// TIA Portal project "PLC_Working" (V16)

(* hardware
DEVICE "S71500/ET200MP station_1"  S7-1500 station
   slot 0: "Rail_0"  Rack  6ES7 590-1***0-0AA0
   slot 1: "PLC_1"  CPU 1515-2 PN  6ES7 515-2AM02-0AB0  V2.8
      slot 3: "CPU display_1"  6ES7591-1BA00-0AA0
      slot 32768: "PROFINET interface_1"  X1
         slot 32769: "Port_1"  X1 P1
         slot 32770: "Port_2"  X1 P2
      slot 33024: "PROFINET interface_2"  X2
      slot 34817: "Virtual CP interface port_1"  Virtual CP interface port  Virtual CP interface port
*)

// ===== PLC "PLC_1"  CPU 1515-2 PN =====

VAR_GLOBAL   // PLC tag table "Default tag table"
   "System_Byte" AT %MB1 : Byte;
   "FirstScan" AT %M1.0 : Bool;
   "DiagStatusUpdate" AT %M1.1 : Bool;
   "AlwaysTRUE" AT %M1.2 : Bool;
   "AlwaysFALSE" AT %M1.3 : Bool;
   "Clock_Byte" AT %MB0 : Byte;
   "Clock_10Hz" AT %M0.0 : Bool;
   "Clock_5Hz" AT %M0.1 : Bool;
   "Clock_2.5Hz" AT %M0.2 : Bool;
   "Clock_2Hz" AT %M0.3 : Bool;
   "Clock_1.25Hz" AT %M0.4 : Bool;
   "Clock_1Hz" AT %M0.5 : Bool;
   "Clock_0.625Hz" AT %M0.6 : Bool;
   "Clock_0.5Hz" AT %M0.7 : Bool;
   "in1" AT %M2.0 : Bool;
   "out1" AT %M2.1 : Bool;
   "out2" AT %M2.2 : Bool;
   "out3" AT %M2.3 : Bool;
   "out3_count" AT %MW4 : Int;
   "out1_count" AT %MW6 : Int;
   "T1_OUT" AT %M2.4 : Bool;
   "T2_OUT" AT %M2.5 : Bool;
   "T3_OUT" AT %M2.6 : Bool;
   "T4_OUT" AT %M2.7 : Bool;
   "ET1" AT %MD8 : Time;
   "ET2" AT %MD12 : Time;
   "ET3" AT %MD16 : DWord;
   "ET4" AT %MD20 : DInt;
   "TIMER_SWITCH" AT %M3.0 : Bool;
   "T4_RESET" AT %M3.1 : Bool;
   "in1 timer" AT %M3.2 : Bool;
END_VAR

DATA_BLOCK "LADDER2_DB"   // DB1
{ S7_Optimized_Access := 'TRUE' }
VERSION : 0.1
// stored: InstanceOfName LADDER2
"LADDER2"
BEGIN
END_DATA_BLOCK

DATA_BLOCK "TIMER_OPERATION_DB"   // DB8
{ S7_Optimized_Access := 'TRUE' }
VERSION : 0.1
// stored: InstanceOfName TIMER_OPERATION
"TIMER_OPERATION"
BEGIN
END_DATA_BLOCK

// folder: System blocks/Program resources

DATA_BLOCK "PULSE_TIMER"   // DB2
{ S7_Optimized_Access := 'TRUE' }
AUTHOR : Simatic
FAMILY : IEC
NAME : IEC_TMR
VERSION : 1.0
// stored: InstanceOfName IEC_TIMER
"IEC_TIMER"
BEGIN
END_DATA_BLOCK

DATA_BLOCK "IEC_Counter_0_DB"   // DB3
{ S7_Optimized_Access := 'TRUE' }
AUTHOR : Simatic
FAMILY : IEC
NAME : CNTR
VERSION : 1.0
// stored: InstanceOfName IEC_COUNTER
"IEC_COUNTER"
BEGIN
END_DATA_BLOCK

DATA_BLOCK "IEC_Counter_0_DB_1"   // DB4
{ S7_Optimized_Access := 'TRUE' }
AUTHOR : Simatic
FAMILY : IEC
NAME : CNTR
VERSION : 1.0
// stored: InstanceOfName IEC_COUNTER
"IEC_COUNTER"
BEGIN
END_DATA_BLOCK

DATA_BLOCK "TON_TIMER"   // DB5
{ S7_Optimized_Access := 'TRUE' }
AUTHOR : Simatic
FAMILY : IEC
NAME : IEC_TMR
VERSION : 1.0
// stored: InstanceOfName IEC_TIMER
"IEC_TIMER"
BEGIN
END_DATA_BLOCK

DATA_BLOCK "TOF_TIMER"   // DB6
{ S7_Optimized_Access := 'TRUE' }
AUTHOR : Simatic
FAMILY : IEC
NAME : IEC_TMR
VERSION : 1.0
// stored: InstanceOfName IEC_TIMER
"IEC_TIMER"
BEGIN
END_DATA_BLOCK

DATA_BLOCK "TONR_TIMER"   // DB7
{ S7_Optimized_Access := 'TRUE' }
AUTHOR : Simatic
FAMILY : IEC
NAME : IEC_TMR
VERSION : 1.0
// stored: InstanceOfName IEC_TIMER
"IEC_TIMER"
BEGIN
END_DATA_BLOCK

// folder: (top level)

FUNCTION_BLOCK "LADDER2"   // FB1, LAD
{ S7_Optimized_Access := 'TRUE' }
VERSION : 0.1
   VAR
      ons : Bool;
   END_VAR
   VAR_TEMP   // added for the SCL form of the ladder/FBD networks
      _w1 : Bool;
   END_VAR
BEGIN

REGION Network 1: device 1 control
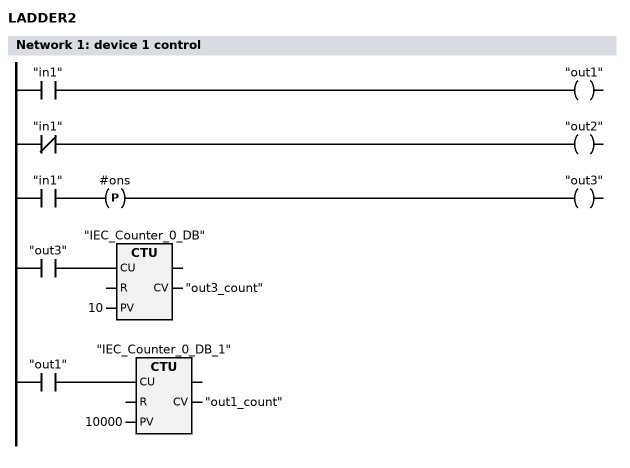
   "out1" := "in1";
   "out2" := NOT "in1";
   #_w1 := "in1" AND NOT #ons;   // rising edge
   #ons := "in1";
   "out3" := #_w1;
   "IEC_Counter_0_DB".CTU(CU := "out3", PV := 10, CV => "out3_count");
   "IEC_Counter_0_DB_1".CTU(CU := "out1", PV := 10000, CV => "out1_count");
END_REGION
END_FUNCTION_BLOCK

FUNCTION_BLOCK "TIMER_OPERATION"   // FB2, LAD
{ S7_Optimized_Access := 'TRUE' }
VERSION : 0.1
BEGIN

REGION Network 1
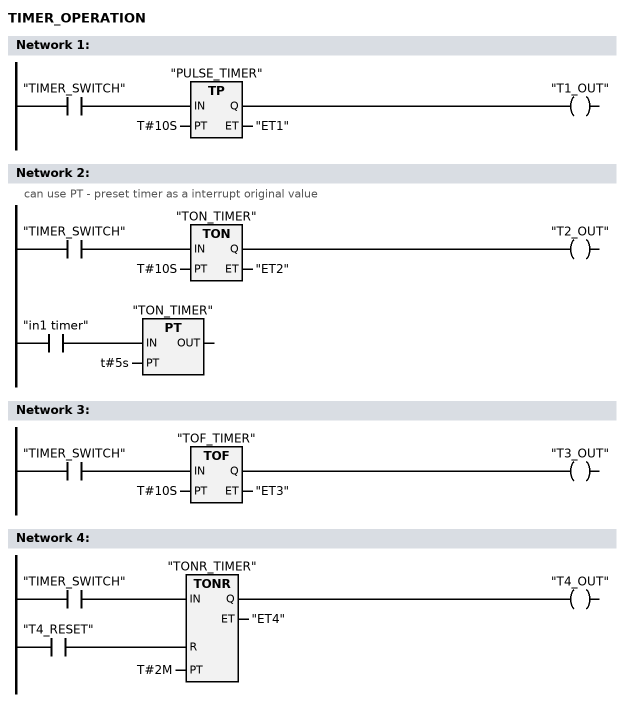
   "PULSE_TIMER".TP(IN := "TIMER_SWITCH", PT := T#10S, ET => "ET1");
   "T1_OUT" := "PULSE_TIMER".Q;
END_REGION

REGION Network 2
   // can use PT - preset timer as a interrupt original value
   "TON_TIMER".TON(IN := "TIMER_SWITCH", PT := T#10S, ET => "ET2");
   "T2_OUT" := "TON_TIMER".Q;
   IF "in1 timer" THEN PRESET_TIMER(PT := t#5s, TIMER := "TON_TIMER"); END_IF;
END_REGION

REGION Network 3
   "TOF_TIMER".TOF(IN := "TIMER_SWITCH", PT := T#10S, ET => "ET3");
   "T3_OUT" := "TOF_TIMER".Q;
END_REGION

REGION Network 4
   "TONR_TIMER".TONR(IN := "TIMER_SWITCH", R := "T4_RESET", PT := T#2M, ET => "ET4");
   "T4_OUT" := "TONR_TIMER".Q;
END_REGION
END_FUNCTION_BLOCK

ORGANIZATION_BLOCK "Main"   // OB1, LAD, ProgramCycle
TITLE = "Main Program Sweep (Cycle)"
{ S7_Optimized_Access := 'TRUE' }
VERSION : 0.1
   VAR_INPUT
      Initial_Call : Bool;   // Initial call of this OB
      Remanence : Bool;   // =True, if remanent data are available
   END_VAR
BEGIN

REGION Network 1
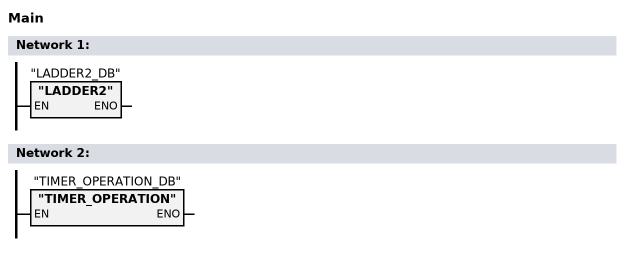
   RUNG wire#powerrail
      "LADDER2_DB"()
   END_RUNG
   // the same network as SCL:
   "LADDER2_DB"();   // "LADDER2"
END_REGION

REGION Network 2
   RUNG wire#powerrail
      "TIMER_OPERATION_DB"()
   END_RUNG
   // the same network as SCL:
   "TIMER_OPERATION_DB"();   // "TIMER_OPERATION"
END_REGION
END_ORGANIZATION_BLOCK